(* IEC 61131-3 sources: Summary-ETFA22/ahorn/benchmark/Arcade, 15 files *)

(* ---- 4.4.SafeMotionIO.st ---- *)
PROGRAM SafeMotionIO
USING PLCopenX;

  VAR_INPUT
	S1_S_EStopIn : SAFEBOOL;
    S2_S_AutoMode : SAFEBOOL;
    S2_S_SetupMode : SAFEBOOL;
    S4_S_EnableSwitchCh1 : SAFEBOOL;
    S4_S_EnableSwitchCh2 : SAFEBOOL;
    S5_S_GuardSwitch : SAFEBOOL;
    S7_S_GuardLock : SAFEBOOL;
    S0_Reset : BOOL;
    S8_UnlockGuard : BOOL;
    M1_S_AcknowledgeSS1 : SAFEBOOL;
    M1_S_AcknowledgeSafeMotion : SAFEBOOL;
  END_VAR
  VAR_OUTPUT
    S_SafeStop_M1 : SAFEBOOL;
    S_SafeMotion_M1 : SAFEBOOL;
    S_Enable_M1 : SAFEBOOL;
    S_UnlockGuard_K1 : SAFEBOOL;
  END_VAR
  VAR
    S_SetupMode : SAFEBOOL;
    S_AutoMode : SAFEBOOL;
    S_SafeStandstill : SAFEBOOL;
    S_SafeMotionActive : SAFEBOOL;
    SF_EmergencyStop_1 : SF_EmergencyStopX;
  	SF_SafetyRequest_1 : SF_SafetyRequestX;
  	SF_SafetyRequest_2 : SafetyRequest_dummy;
  	SF_ModeSelector_1 : SF_ModeSelectorX;
  	SF_GuardLocking_1 : SF_GuardLockingX;
  	SF_EnableSwitch_1 : SF_EnableSwitchX;
  END_VAR

  SF_EmergencyStop_1(TRUE, S1_S_EStopIn, FALSE, FALSE, S0_Reset);
  SF_SafetyRequest_1(TRUE, SF_EmergencyStop_1.S_EstopOut, M1_S_AcknowledgeSS1, T#100ms, S0_Reset);
  SF_SafetyRequest_2(TRUE, S_AutoMode, M1_S_AcknowledgeSafeMotion, T#100ms, S0_Reset);
  SF_ModeSelector_1(TRUE, S2_S_AutoMode, S2_S_SetupMode, FALSE, FALSE, FALSE, FALSE, FALSE, FALSE, TRUE, FALSE, TRUE, T#50ms, S0_Reset);
  SF_GuardLocking_1(TRUE, S5_S_GuardSwitch, S_SafeStandstill OR S_SafeMotionActive, S7_S_GuardLock, S8_UnlockGuard, FALSE, FALSE, S0_Reset);
  SF_EnableSwitch_1(TRUE, S_SafeMotionActive AND S_SetupMode, S4_S_EnableSwitchCh1, S4_S_EnableSwitchCh2, FALSE, S0_Reset);

  S_SafeStandstill := SF_SafetyRequest_1.S_SafetyActive;
  S_SafeStop_M1 := SF_SafetyRequest_1.S_SafetyRequest;
  S_SafeMotionActive := SF_SafetyRequest_2.S_SafetyActive;
  S_SafeMotion_M1 := SF_SafetyRequest_2.S_SafetyRequest;
  S_SetupMode := SF_ModeSelector_1.S_Mode1Sel;
  S_AutoMode := SF_ModeSelector_1.S_Mode0Sel AND SF_GuardLocking_1.S_GuardLocked;
  S_UnlockGuard_K1 := SF_GuardLocking_1.S_UnlockGuard;
  S_Enable_M1 := SF_EnableSwitch_1.S_EnableSwitchOut;

END_PROGRAM

FUNCTION_BLOCK SafetyRequest_dummy
VAR_INPUT
        Activate        : BOOL;
        S_OpMode        : SAFEBOOL;
        S_Acknowledge   : SAFEBOOL;
        MonitoringTime  : TIME := T#0s;
        Reset           : BOOL ;
 END_VAR

 VAR_OUTPUT
        Ready : BOOL ;
        S_SafetyActive : SAFEBOOL ;
        S_SafetyRequest : SAFEBOOL ;
        Error : BOOL ;
        DiagCode : WORD:=16#0000 ;
 END_VAR

VAR
        R_TRIGatReset: R_TRIG;
        T1: TONX;
END_VAR

R_TRIGatReset(CLK:=Reset);

IF NOT Activate THEN
    DiagCode := 16#0000;
ELSE

CASE DiagCode OF
16#0000:
    IF Activate THEN
        DiagCode := 16#8001;
    END_IF;
16#8000:
    IF NOT S_Acknowledge THEN
        DiagCode := 16#C002;
    ELSIF S_OpMode THEN
        DiagCode := 16#8012;
    END_IF;
16#8001:
    IF R_TRIGatReset.Q AND NOT S_Acknowledge THEN
        DiagCode := 16#8002;
    ELSIF R_TRIGatReset.Q AND S_Acknowledge THEN
        DiagCode := 16#8012;
    END_IF;
16#8002:
    IF NOT S_OpMode THEN
        DiagCode := 16#8003;
    ELSIF S_Acknowledge THEN
        DiagCode := 16#8012;
    END_IF;
16#8003:
    IF T1.Q THEN
        DiagCode := 16#C003;
    ELSIF S_OpMode THEN
        DiagCode := 16#8012;
    ELSIF S_Acknowledge THEN
        DiagCode := 16#8000;
    END_IF;
16#8005:
    IF S_OpMode THEN
        DiagCode := 16#8012;
    END_IF;
16#8012:
    IF NOT S_Acknowledge THEN
        DiagCode := 16#8002;
    ELSIF NOT S_OpMode THEN
        DiagCode := 16#8003;
    END_IF;
16#C002:
    IF Reset AND NOT R_TRIGatReset.Q THEN
        DiagCode := 16#C004;
    ELSIF R_TRIGatReset.Q THEN
        DiagCode := 16#8005;
    END_IF;
16#C003:
    IF Reset AND NOT R_TRIGatReset.Q THEN
        DiagCode := 16#C005;
    ELSIF R_TRIGatReset.Q THEN
        DiagCode := 16#8005;
    END_IF;
16#C004:
    IF NOT Reset THEN
        DiagCode := 16#C002;
    END_IF;
16#C005:
    IF NOT Reset THEN
        DiagCode := 16#C003;
    END_IF;
END_CASE;
END_IF;

IF DiagCode <> 16#8003 THEN
    T1(IN:=false, PT:=MonitoringTime);
ELSE
	T1(IN:=true, PT:=MonitoringTime);
END_IF;

CASE DiagCode OF
16#0000:
    Ready := FALSE;
    S_SafetyActive := FALSE;
    S_SafetyRequest := FALSE;
    Error := FALSE;
16#8000:
    Ready := TRUE;
    S_SafetyActive := TRUE;
    S_SafetyRequest := FALSE;
    Error := FALSE;
16#8001:
    Ready := TRUE;
    S_SafetyActive := FALSE;
    S_SafetyRequest := FALSE;
    Error := FALSE;
16#8002:
    Ready := TRUE;
    S_SafetyActive := FALSE;
    S_SafetyRequest := TRUE;
    Error := FALSE;
16#8003:
    Ready := TRUE;
    S_SafetyActive := FALSE;
    S_SafetyRequest := FALSE;
    Error := FALSE;
16#8005:
    Ready := TRUE;
    S_SafetyActive := FALSE;
    S_SafetyRequest := FALSE;
    Error := FALSE;
16#8012:
    Ready := TRUE;
    S_SafetyActive := FALSE;
    S_SafetyRequest := TRUE;
    Error := FALSE;
16#C002:
    Ready := TRUE;
    S_SafetyActive := FALSE;
    S_SafetyRequest := FALSE;
    Error := TRUE;
16#C003:
    Ready := TRUE;
    S_SafetyActive := FALSE;
    S_SafetyRequest := FALSE;
    Error := TRUE;
16#C004:
    Ready := TRUE;
    S_SafetyActive := FALSE;
    S_SafetyRequest := FALSE;
    Error := TRUE;
16#C005:
    Ready := TRUE;
    S_SafetyActive := FALSE;
    S_SafetyRequest := FALSE;
    Error := TRUE;
END_CASE;

END_FUNCTION_BLOCK;

(* ---- antivalentX.st ---- *)
FUNCTION_BLOCK SF_Antivalent2
 VAR_INPUT
        Activate           : BOOL;
        S_ChannelNC        : SAFEBOOL;
        S_ChannelNO        : SAFEBOOL;
        DiscrepancyTime    : TIME;
 END_VAR
 VAR_OUTPUT
        Ready              : BOOL;
        S_AntivalentOut    : BOOL;
        Error              : BOOL;
        DiagCode           : WORD;
 END_VAR
 VAR
        T_1        : TONX;
 END_VAR

IF NOT Activate THEN
    DiagCode := 16#0000;
ELSE

CASE DiagCode OF
16#0000:
    IF Activate THEN
        DiagCode := 16#8001;
    END_IF;
16#8001:
    IF S_ChannelNC AND S_ChannelNO THEN
        DiagCode := 16#8004;
        T_1(IN:=1, PT:=DiscrepancyTime);
    ELSIF NOT S_ChannelNC AND NOT S_ChannelNO THEN
        DiagCode := 16#8014;
        T_1(IN:=1, PT:=DiscrepancyTime);
    ELSIF S_ChannelNC AND NOT S_ChannelNO THEN
        DiagCode := 16#8000;
    END_IF;
16#8004:
    IF T_1.Q THEN
        DiagCode := 16#C001;
    ELSIF NOT S_ChannelNC THEN
        DiagCode := 16#8001;
    ELSIF NOT S_ChannelNO THEN
        DiagCode := 16#8000;
    END_IF;
16#C001,
16#C002:
    IF NOT S_ChannelNC AND S_ChannelNO THEN
        DiagCode := 16#8001;
    END_IF;
16#8014:
    IF T_1.Q THEN
        DiagCode := 16#C002;
    ELSIF S_ChannelNO THEN
        DiagCode := 16#8001;
    ELSIF S_ChannelNC THEN
        DiagCode := 16#8000;
    END_IF;
16#C003:
    IF NOT S_ChannelNC AND S_ChannelNO THEN
        DiagCode := 16#8001;
    END_IF;
16#8005:
    IF T_1.Q THEN
        DiagCode := 16#C003;
    ELSIF NOT S_ChannelNC AND S_ChannelNO THEN
        DiagCode := 16#8001;
    END_IF;
16#8000:
    IF NOT S_ChannelNC OR S_ChannelNO THEN
        DiagCode := 16#8005;
        T_1(IN:=1, PT:=DiscrepancyTime);
    ELSIF NOT S_ChannelNC AND S_ChannelNO THEN
        DiagCode := 16#8001;
    END_IF;
END_CASE;
END_IF;

CASE DiagCode OF
16#0000:
    T_1(IN:=0, PT:=DiscrepancyTime);
    Ready := FALSE;
    Error := FALSE;
    S_AntivalentOut:= FALSE;
16#8000:
    T_1(IN:=0, PT:=DiscrepancyTime);
    Ready := TRUE;
    Error := FALSE;
    S_AntivalentOut := TRUE;
16#8001:
    T_1(IN:=0, PT:=DiscrepancyTime);
    Ready := TRUE;
    Error := FALSE;
    S_AntivalentOut:= FALSE;
16#8004,
16#8014,
16#8005:
	T_1(IN:=1, PT:=DiscrepancyTime);
    Ready := TRUE;
    Error := FALSE;
    S_AntivalentOut:= FALSE;
16#C001,
16#C002,
16#C003:
    T_1(IN:=0, PT:=DiscrepancyTime);
    Ready := TRUE;
    Error := TRUE;
    S_AntivalentOut:= FALSE;
END_CASE;

END_FUNCTION_BLOCK

(* ---- emergencyStopX.st ---- *)
FUNCTION_BLOCK SF_EmergencyStop2
VAR_INPUT
        Activate      : BOOL;
        S_EStopIn     : BOOL;
        S_StartReset  : BOOL;
        S_AutoReset   : BOOL;
        Reset         : BOOL;
 END_VAR

 VAR_OUTPUT
        Ready         : BOOL;
        S_EStopOut    : BOOL;
        Error         : BOOL;
        DiagCode      : WORD;
 END_VAR

 VAR
        R_TRIGatReset: R_TRIG;
 END_VAR

R_TRIGatReset(CLK:=Reset);

IF NOT Activate THEN
    DiagCode := 16#0000;
ELSE

CASE DiagCode OF
16#0000:
    IF Activate THEN
        DiagCode := 16#8001;
    END_IF;
16#8001:
    IF NOT S_StartReset THEN
        DiagCode := 16#8002;
    ELSIF S_StartReset AND NOT S_EStopIn THEN
        DiagCode := 16#8004;
    ELSIF S_EStopIn AND S_StartReset THEN
        DiagCode := 16#8000;
    END_IF;
16#8002:
    IF S_EStopIn THEN
        DiagCode := 16#8003;
    END_IF;
16#8003:
    IF Reset AND NOT R_TRIGatReset.Q THEN
        DiagCode := 16#C001;
    ELSIF NOT S_EStopIn THEN
        DiagCode := 16#8002;
    ELSIF R_TRIGatReset.Q THEN
        DiagCode := 16#8000;
    END_IF;
16#C001:
    IF NOT Reset THEN
        DiagCode := 16#8003;
    END_IF;
16#8004:
    IF S_EStopIn AND NOT S_AutoReset THEN
        DiagCode := 16#8005;
    ELSIF S_EStopIn AND S_AutoReset THEN
        DiagCode := 16#8000;
    END_IF;
16#8005:
    IF Reset AND NOT R_TRIGatReset.Q THEN
        DiagCode := 16#C002;
    ELSIF NOT S_EStopIn THEN
        DiagCode := 16#8004;
    ELSIF R_TRIGatReset.Q OR S_AutoReset THEN
        DiagCode := 16#8000;
    END_IF;
16#C002:
    IF NOT Reset THEN
        DiagCode := 16#8005;
    END_IF;
16#8000:
    IF NOT S_EStopIn THEN
        DiagCode := 16#8004;
    END_IF;
END_CASE;
END_IF;

CASE DiagCode OF
16#0000:
    Ready := FALSE;
    Error := FALSE;
    S_EStopOut := FALSE;
16#8001:
    Ready := TRUE;
    Error := FALSE;
    S_EStopOut := FALSE;
16#8002:
    Ready := TRUE;
    Error := FALSE;
    S_EStopOut := FALSE;
16#8003:
    Ready := TRUE;
    Error := FALSE;
    S_EStopOut := FALSE;
16#C001:
    Ready := TRUE;
    Error := TRUE;
    S_EStopOut := FALSE;
16#8004:
    Ready := TRUE;
    Error := FALSE;
    S_EStopOut := FALSE;
16#8005:
    Ready := TRUE;
    Error := FALSE;
    S_EStopOut := FALSE;
16#C002:
    Ready := TRUE;
    Error := TRUE;
    S_EStopOut := FALSE;
16#8000:
    Ready := TRUE;
    Error := FALSE;
    S_EStopOut := TRUE;
END_CASE;

END_FUNCTION_BLOCK

(* ---- enableSwitchX.st ---- *)
FUNCTION_BLOCK SF_EnableSwitch2
VAR_INPUT
	Activate          : BOOL := FALSE;
	S_SafetyActive    : SAFEBOOL := FALSE;
	S_EnableSwitchCh1 : SAFEBOOL := FALSE;
	S_EnableSwitchCh2 : SAFEBOOL := FALSE;
	S_AutoReset       : SAFEBOOL := FALSE;
	Reset             : BOOL := FALSE;
END_VAR

VAR_OUTPUT
	Ready: BOOL := FALSE;
	S_EnableSwitchOut: SAFEBOOL := FALSE;
	Error: BOOL := FALSE;
	DiagCode: WORD := 16#0000;
END_VAR

VAR
	R_TRIGatReset: R_TRIG;
END_VAR

R_TRIGatReset(CLK:=Reset);

IF NOT Activate THEN
    DiagCode := 16#0000;
ELSIF NOT S_SafetyActive THEN
    DiagCode := 16#8004;
ELSE

CASE DiagCode OF
16#0000:
    IF Activate THEN
	DiagCode := 16#8004;
    END_IF;

16#8000:
	IF (NOT (S_EnableSwitchCh1 OR S_EnableSwitchCh2)) OR (S_EnableSwitchCh1 AND NOT S_EnableSwitchCh2) THEN
		DiagCode := 16#8007;
	ELSIF NOT S_EnableSwitchCh1 AND S_EnableSwitchCh2 THEN
		DiagCode := 16#8006;
	END_IF;

16#8004:
    IF S_SafetyActive THEN
		DiagCode := 16#8005;
	END_IF;

16#8005:
	IF NOT (NOT S_EnableSwitchCh1 AND S_EnableSwitchCh2) THEN
		DiagCode := 16#C010;
	ELSIF NOT S_EnableSwitchCh1 AND S_EnableSwitchCh2 THEN
		DiagCode := 16#8006;
	END_IF;

16#8006:
	IF S_EnableSwitchCh1 AND S_EnableSwitchCh2 THEN
		DiagCode := 16#8000;
	ELSIF (NOT (S_EnableSwitchCh1 OR S_EnableSwitchCh2)) OR (S_EnableSwitchCh1 AND NOT S_EnableSwitchCh2) THEN
		DiagCode := 16#8007;
	END_IF;

16#8007:
	IF S_EnableSwitchCh1 AND S_EnableSwitchCh2 THEN
		DiagCode := 16#C030;
	ELSIF NOT S_EnableSwitchCh1 AND S_EnableSwitchCh2 THEN
		DiagCode := 16#8006;
	END_IF;
16#C001:
	IF NOT Reset THEN
		DiagCode := 16#C020;
	END_IF;
16#C002:
	IF NOT Reset THEN
		DiagCode := 16#C040;
	END_IF;
16#C010:
	IF NOT S_EnableSwitchCh1 AND S_EnableSwitchCh2 THEN
		DiagCode := 16#C020;
	END_IF;

16#C020:
	IF NOT (NOT S_EnableSwitchCh1 AND S_EnableSwitchCh2) THEN
		DiagCode := 16#C010;
	ELSIF Reset AND NOT R_TRIGatReset.Q AND NOT S_AutoReset THEN
		DiagCode := 16#C001;
	ELSIF R_TRIGatReset.Q OR S_AutoReset THEN
		DiagCode := 16#8006;
	END_IF;

16#C030:
	IF NOT (S_EnableSwitchCh1 AND S_EnableSwitchCh2) THEN
		DiagCode := 16#C040;
	END_IF;

16#C040:
	IF S_EnableSwitchCh1 AND S_EnableSwitchCh2 THEN
		DiagCode := 16#C030;
	ELSIF Reset AND R_TRIGatReset.Q AND NOT S_AutoReset THEN
		DiagCode := 16#C002;
	ELSIF R_TRIGatReset.Q OR S_AutoReset THEN
		DiagCode := 16#8007;
	END_IF;
END_CASE;

END_IF;

CASE DiagCode OF
16#C001,
16#C002,
16#C010,
16#C020,
16#C030,
16#C040:
	Ready := TRUE;
	S_EnableSwitchOut := FALSE;
	Error := TRUE;
16#0000:
	Ready := FALSE;
	S_EnableSwitchOut := FALSE;
	Error := FALSE;
16#8000:
	Ready := TRUE;
	S_EnableSwitchOut := TRUE;
	Error := FALSE;

16#8004,
16#8005,
16#8006,
16#8007:
	Ready := TRUE;
	S_EnableSwitchOut := FALSE;
	Error := FALSE;

END_CASE;

END_FUNCTION_BLOCK

(* ---- equivalentX.st ---- *)
FUNCTION_BLOCK equivalentX
VAR_INPUT
	Activate		: BOOL;
	S_ChannelA		: BOOL;
	S_ChannelB		: BOOL;
	DiscrepancyTime 	: TIME;
END_VAR
VAR_OUTPUT
	Ready		: BOOL;
	S_EquivalentOut	: BOOL;
	Error		: BOOL;
	DiagCode	: WORD;
END_VAR
VAR
 DiscrepancyTimer	: TONX;
END_VAR

IF NOT Activate THEN
    DiagCode := 16#0000;
ELSE

CASE DiagCode OF
16#0000:
    IF Activate THEN
	DiagCode := 16#8001;
    END_IF;
16#8001:
    IF S_ChannelA AND NOT S_ChannelB THEN
	DiagCode := 16#8004;
    ELSIF S_ChannelB AND NOT S_ChannelA THEN
	DiagCode := 16#8014;
    ELSIF S_ChannelA AND S_ChannelB THEN
	DiagCode := 16#8000;
    END_IF;
16#8004:
    IF DiscrepancyTimer.Q THEN
	DiagCode := 16#C001;
    ELSIF NOT S_ChannelA THEN
	DiagCode := 16#8001;
    ELSIF S_ChannelB THEN
	DiagCode := 16#8000;
    END_IF;
16#C001,
16#C002:
    IF NOT S_ChannelA AND NOT S_ChannelB THEN
	DiagCode := 16#8001;
    END_IF;
16#8014:
    IF DiscrepancyTimer.Q THEN
	DiagCode := 16#C002;
    ELSIF NOT S_ChannelB THEN
	DiagCode := 16#8001;
    ELSIF S_ChannelA THEN
	DiagCode := 16#8000;
    END_IF;
16#C003:
    IF NOT S_ChannelA AND NOT S_ChannelB THEN
	DiagCode := 16#8001;
    END_IF;
16#8005:
    IF DiscrepancyTimer.Q THEN
	DiagCode := 16#C003;
    ELSIF NOT S_ChannelA AND NOT S_ChannelB THEN
	DiagCode := 16#8001;
    END_IF;
16#8000:
    IF S_ChannelA XOR S_ChannelB THEN
	DiagCode := 16#8005;
    ELSIF NOT S_ChannelA AND NOT S_ChannelB THEN
	DiagCode := 16#8001;
    END_IF;
END_CASE;

END_IF;

CASE DiagCode OF
16#0000:
    DiscrepancyTimer(IN:=0, PT:=DiscrepancyTime);
    Ready := FALSE;
    Error := FALSE;
    S_EquivalentOut:= FALSE;
16#8000:
    DiscrepancyTimer(IN:=0, PT:=DiscrepancyTime);
    Ready := TRUE;
    Error := FALSE;
    S_EquivalentOut := TRUE;
16#8001:
    DiscrepancyTimer(IN:=0, PT:=DiscrepancyTime);
    Ready := TRUE;
    Error := FALSE;
    S_EquivalentOut:= FALSE;
16#8004,
16#8014,
16#8005:
	DiscrepancyTimer(IN:=1, PT:=DiscrepancyTime);
    Ready := TRUE;
    Error := FALSE;
    S_EquivalentOut:= FALSE;
16#C001,
16#C002,
16#C003:
    DiscrepancyTimer(IN:=0, PT:=DiscrepancyTime);
    Ready := TRUE;
    Error := TRUE;
    S_EquivalentOut:= FALSE;
END_CASE;

END_FUNCTION_BLOCK

(* ---- guardLockingX.st ---- *)
FUNCTION_BLOCK SF_GuardLocking2
VAR_INPUT
        Activate          : BOOL;
        S_GuardMonitoring : SAFEBOOL;
        S_SafetyActive    : SAFEBOOL;
        S_GuardLock       : SAFEBOOL;
        UnlockRequest     : BOOL;
        S_StartReset      : SAFEBOOL;
        S_AutoReset       : SAFEBOOL;
        Reset             : BOOL;
 END_VAR

 VAR_OUTPUT
    Ready             : BOOL;
    S_GuardLocked     : SAFEBOOL;
    S_UnlockGuard     : SAFEBOOL;
    Error             : BOOL;
         DiagCode                  : WORD:=16#0000;
 END_VAR

VAR
        R_TRIGatReset: R_TRIG;
        R_TRIGatUnlockRequest: R_TRIG;
END_VAR

R_TRIGatReset(CLK:=Reset);
R_TRIGatUnlockRequest(CLK:=UnlockRequest);

IF NOT Activate THEN
    DiagCode := 16#0000;
END_IF;

CASE DiagCode OF
16#0000:
    IF Activate THEN
        DiagCode := 16#8001;
    END_IF;
16#8000:
    IF NOT S_GuardLock OR NOT S_GuardMonitoring THEN
        DiagCode := 16#C004;
    ELSIF R_TRIGatUnlockRequest.Q AND S_SafetyActive THEN
        DiagCode := 16#8013;
    END_IF;
16#8001:
    IF Reset AND NOT R_TRIGatReset.Q AND NOT S_StartReset THEN
        DiagCode := 16#C001;
    ELSIF NOT S_GuardLock OR NOT S_GuardMonitoring THEN
        DiagCode := 16#8011;
    ELSIF (R_TRIGatReset.Q OR S_StartReset) AND S_GuardMonitoring AND S_GuardLock THEN
        DiagCode := 16#8000;
    END_IF;
16#8003:
    IF Reset AND NOT R_TRIGatReset.Q AND NOT S_AutoReset THEN
        DiagCode := 16#C003;
    ELSIF NOT S_GuardMonitoring OR NOT S_GuardLock THEN
        DiagCode := 16#8011;
    ELSIF R_TRIGatReset.Q OR S_AutoReset THEN
        DiagCode := 16#8000;
    END_IF;
16#8011:
    IF NOT S_SafetyActive AND (NOT S_GuardMonitoring OR NOT S_GuardLock) THEN
        DiagCode := 16#C004;
    ELSIF (S_SafetyActive AND UnlockRequest) OR NOT S_GuardMonitoring THEN
        DiagCode := 16#8012;
    ELSIF S_GuardMonitoring AND S_GuardLock THEN
        DiagCode := 16#8003;
    END_IF;
16#8012:
    IF S_GuardMonitoring THEN
        DiagCode := 16#8013;
    ELSIF NOT S_SafetyActive AND NOT S_GuardMonitoring THEN
        DiagCode := 16#C004;
    END_IF;
16#8013:
    IF NOT S_GuardMonitoring THEN
        DiagCode := 16#8012;
    ELSIF NOT UnlockRequest THEN
        DiagCode := 16#8011;
    END_IF;
16#8014:
    IF Reset AND NOT R_TRIGatReset.Q THEN
        DiagCode := 16#C002;
    ELSIF NOT S_SafetyActive THEN
        DiagCode := 16#C004;
    ELSIF R_TRIGatReset.Q THEN
        DiagCode := 16#8011;
    END_IF;
16#C001:
    IF NOT Reset THEN
        DiagCode := 16#8001;
    END_IF;
16#C002:
    IF NOT Reset THEN
        DiagCode := 16#8014;
    END_IF;
16#C003:
    IF NOT Reset THEN
        DiagCode := 16#8003;
    END_IF;
16#C004:
    IF S_SafetyActive THEN
        DiagCode := 16#8014;
    END_IF;
END_CASE;

CASE DiagCode OF
16#0000:
    Ready := FALSE;
    S_GuardLocked := FALSE;
    S_UnlockGuard := FALSE;
    Error := FALSE;
16#8000:
    Ready := TRUE;
    S_GuardLocked := TRUE;
    S_UnlockGuard := FALSE;
    Error := FALSE;
16#8001,
16#8003,
16#8011,
16#8014:
    Ready := TRUE;
    S_GuardLocked := FALSE;
    S_UnlockGuard := FALSE;
    Error := FALSE;
16#8012,
16#8013:
    Ready := TRUE;
    S_GuardLocked := FALSE;
    S_UnlockGuard := TRUE;
    Error := FALSE;
16#C001,
16#C002,
16#C003,
16#C004:
    Ready := TRUE;
    S_GuardLocked := FALSE;
    S_UnlockGuard := FALSE;
    Error := TRUE;
END_CASE;

END_FUNCTION_BLOCK

(* ---- guardMonitoringX.st ---- *)
FUNCTION_BLOCK SF_GuardMonitoring2
VAR_INPUT
        Activate        : BOOL := FALSE;
        S_GuardSwitch1  : SAFEBOOL := FALSE;
        S_GuardSwitch2  : SAFEBOOL := FALSE;
        DiscrepancyTime : TIME := T#0s;
        S_StartReset    : SAFEBOOL := FALSE;
        S_AutoReset     : SAFEBOOL := FALSE;
        Reset           : BOOL := FALSE;
END_VAR
VAR_OUTPUT
        Ready             : BOOL := FALSE;
        S_GuardMonitoring : BOOL := FALSE;
        Error             : BOOL := FALSE;
        DiagCode          : WORD := 16#0000;
END_VAR
VAR
    R_TRIGatReset : R_TRIG;
    DiscrepancyTimer : TONX;
END_VAR

R_TRIGatReset(CLK:=Reset);

IF NOT Activate THEN
    DiagCode := 16#0000;
ELSE

CASE DiagCode OF
16#0000:
    IF Activate THEN
        DiagCode := 16#8001;
    END_IF;
16#8001:
    IF NOT S_GuardSwitch1 OR NOT S_GuardSwitch2 THEN
        DiagCode := 16#8002;
    ELSIF S_GuardSwitch1 AND S_GuardSwitch2 AND NOT S_StartReset THEN
        DiagCode := 16#8003;
    ELSIF S_GuardSwitch1 AND S_GuardSwitch2 AND S_StartReset THEN
        DiagCode := 16#8000;
    END_IF;
16#8002:
    IF NOT S_GuardSwitch1 AND NOT S_GuardSwitch2 THEN
        DiagCode := 16#8012;
    END_IF;
16#8003:
    IF Reset AND NOT R_TRIGatReset.Q THEN
        DiagCode := 16#C001;
    ELSIF NOT S_GuardSwitch1 OR NOT S_GuardSwitch2 THEN
        DiagCode := 16#8002;
    ELSIF R_TRIGatReset.Q THEN
        DiagCode := 16#8000;
    END_IF;
16#8012:
    IF S_GuardSwitch1 THEN
        DiagCode := 16#8004;
    ELSIF S_GuardSwitch2 THEN
        DiagCode := 16#8014;
    END_IF;
16#8004:
    IF DiscrepancyTimer.Q THEN
        DiagCode := 16#C011;
    ELSIF NOT S_GuardSwitch1 THEN
        DiagCode := 16#8002;
    ELSIF S_GuardSwitch2 THEN
        DiagCode := 16#8005;
    END_IF;
16#8014:
    IF DiscrepancyTimer.Q THEN
        DiagCode := 16#C012;
    ELSIF NOT S_GuardSwitch2 THEN
        DiagCode := 16#8002;
    ELSIF S_GuardSwitch1 THEN
        DiagCode := 16#8005;
    END_IF;
16#8005:
    IF NOT S_GuardSwitch1 OR NOT S_GuardSwitch2 THEN
        DiagCode := 16#8002;
    ELSIF NOT S_AutoReset THEN
        DiagCode := 16#8003;
    ELSIF S_AutoReset THEN
        DiagCode := 16#8000;
    END_IF;
16#8000:
    IF NOT S_GuardSwitch1 OR NOT S_GuardSwitch2 THEN
        DiagCode := 16#8002;
    END_IF;
16#C001:
    IF NOT Reset THEN
        DiagCode := 16#8003;
    END_IF;
16#C011:
    IF NOT S_GuardSwitch1 AND NOT S_GuardSwitch2 THEN
        DiagCode := 16#8012;
    END_IF;
16#C012:
    IF NOT S_GuardSwitch1 AND NOT S_GuardSwitch2 THEN
        DiagCode := 16#8012;
    END_IF;
END_CASE;
END_IF;

CASE DiagCode OF
16#0000:
    DiscrepancyTimer(IN:=FALSE, PT:=DiscrepancyTime);
    Ready := FALSE;
    Error := FALSE;
    S_GuardMonitoring := FALSE;
16#8000:
    DiscrepancyTimer(IN:=FALSE, PT:=DiscrepancyTime);
    Ready := TRUE;
    Error := FALSE;
    S_GuardMonitoring  := TRUE;
16#8001,
16#8002,
16#8003,
16#8012,
16#8005:
    DiscrepancyTimer(IN:=FALSE, PT:=DiscrepancyTime);
    Ready := TRUE;
    Error := FALSE;
    S_GuardMonitoring := FALSE;
16#8004,
16#8014:
	DiscrepancyTimer(IN:=TRUE, PT:=DiscrepancyTime);
    Ready := TRUE;
    Error := FALSE;
    S_GuardMonitoring := FALSE;
16#C001,
16#C011,
16#C012:
    DiscrepancyTimer(IN:=FALSE, PT:=DiscrepancyTime);
    Ready := TRUE;
    Error := TRUE;
    S_GuardMonitoring := FALSE;
END_CASE;

END_FUNCTION_BLOCK

(* ---- ModeSelectorX.st ---- *)
FUNCTION_BLOCK ModeSelectorX
VAR_INPUT
        Activate        : BOOL;
        S_Mode0         : BOOL;
        S_Mode1         : BOOL;
        S_Mode2         : BOOL;
        S_Mode3         : BOOL;
        S_Mode4         : BOOL;
        S_Mode5         : BOOL;
        S_Mode6         : BOOL;
        S_Mode7         : BOOL;
        S_Unlock        : BOOL;
        S_SetMode       : BOOL;
        AutoSetMode     : BOOL;
        ModeMonitorTime : TIME;
        Reset           : BOOL;
 END_VAR
 VAR_OUTPUT
        Ready           : BOOL;
        S_Mode0Sel      : BOOL;
        S_Mode1Sel      : BOOL;
        S_Mode2Sel      : BOOL;
        S_Mode3Sel      : BOOL;
        S_Mode4Sel      : BOOL;
        S_Mode5Sel      : BOOL;
        S_Mode6Sel      : BOOL;
        S_Mode7Sel      : BOOL;
        S_AnyModeSel    : BOOL;
        Error           : BOOL;
        DiagCode        : WORD;
 END_VAR
 VAR
        T_1        : TONX;                 (* Timer for S2, transition T27 *)
 END_VAR

 VAR
        R_TRIGatReset: R_TRIG;
        R_TRIGatSetMode: R_TRIG;
        F_TRIGatModeSel0: F_TRIG;
        R_TRIGatModeSel0: R_TRIG;
        fallingEdgeDetected : BOOL;
 END_VAR

 VAR_TEMP
    Error1 : BOOL;
    Error2 : BOOL;
 END_VAR

R_TRIGatReset(CLK:=Reset);
R_TRIGatSetMode(CLK:=S_SetMode);

IF NOT Activate THEN
    DiagCode := 16#0000;
ELSE

IF (S_Mode0 + S_Mode1 + S_Mode2 + S_Mode3 + S_Mode4 + S_Mode5 + S_Mode6 + S_Mode7 > 1) THEN
    Error1 := true;
ELSE
    Error1 := false;
END_IF;

CASE DiagCode OF
16#0000:
    IF Activate THEN
        DiagCode := 16#8005;
    END_IF;
16#8005:
    IF (NOT S_Mode0 AND NOT S_Mode1 AND NOT S_Mode2 AND NOT S_Mode3 AND NOT S_Mode4 AND NOT S_Mode5 AND NOT S_Mode6 AND NOT S_Mode7) THEN
        F_TRIGatModeSel0(CLK:=false);
        R_TRIGatModeSel0(CLK:=false);
    ELSE
        F_TRIGatModeSel0(CLK:=true);
        R_TRIGatModeSel0(CLK:=true);
    END_IF;

    IF F_TRIGatModeSel0.Q THEN
        fallingEdgeDetected := TRUE;
    END_IF;

    IF fallingEdgeDetected THEN
        T_1(IN:=true, PT:=ModeMonitorTime);
    ELSIF R_TRIGatModeSel0.Q THEN
        T_1(IN:=false, PT:=ModeMonitorTime);
        fallingEdgeDetected := FALSE;
    END_IF;

    Error2 := T_1.Q;

    IF Error1 THEN
        DiagCode := 16#C001;
    ELSIF Error2 THEN
        DiagCode := 16#C002;
    ELSIF ((AutoSetMode OR R_TRIGatSetMode.Q) AND S_Unlock AND (S_Mode0 + S_Mode1 + S_Mode2 + S_Mode3 + S_Mode4 + S_Mode5 + S_Mode6 + S_Mode7 = 1)) THEN
        DiagCode := 16#8000;
    END_IF;
16#8000:
    IF Error1 THEN
        DiagCode := 16#C001;
    ELSIF (S_Mode0 <> S_Mode0Sel OR S_Mode1 <> S_Mode1Sel OR S_Mode2 <> S_Mode2Sel OR S_Mode3 <> S_Mode3Sel
          OR S_Mode4 <> S_Mode4Sel OR S_Mode5 <> S_Mode5Sel OR S_Mode6 <> S_Mode6Sel OR S_Mode7 <> S_Mode7Sel) THEN
        DiagCode := 16#8005;
        fallingEdgeDetected := FALSE;
    ELSIF (NOT S_Unlock) THEN
        DiagCode := 16#8004;
    END_IF;
16#8004:
    IF S_Unlock THEN
        DiagCode := 16#8000;
    END_IF;
16#C001:
    IF Reset AND NOT R_TRIGatReset.Q THEN
        DiagCode := 16#C003;
    ELSIF R_TRIGatReset.Q THEN
        DiagCode := 16#8005;
        fallingEdgeDetected := FALSE;
    END_IF;
16#C002:
    IF Reset AND NOT R_TRIGatReset.Q THEN
        DiagCode := 16#C004;
    ELSIF R_TRIGatReset.Q THEN
        DiagCode := 16#8005;
        fallingEdgeDetected := FALSE;
    END_IF;
16#C003:
    IF (NOT Reset) THEN
                DiagCode := 16#C001;
    END_IF;
16#C004:
    IF (NOT Reset) THEN
                DiagCode := 16#C002;
    END_IF;
END_CASE;
END_IF;

CASE DiagCode OF
16#0000:
    Ready := false;
    S_Mode0Sel := false;
    S_Mode1Sel := false;
    S_Mode2Sel := false;
    S_Mode3Sel := false;
    S_Mode4Sel := false;
    S_Mode5Sel := false;
    S_Mode6Sel := false;
    S_Mode7Sel := false;
    S_AnyModeSel := false;
    Error := false;
16#8005:
    Ready := true;
    S_Mode0Sel := false;
    S_Mode1Sel := false;
    S_Mode2Sel := false;
    S_Mode3Sel := false;
    S_Mode4Sel := false;
    S_Mode5Sel := false;
    S_Mode6Sel := false;
    S_Mode7Sel := false;
    S_AnyModeSel := false;
    Error := false;
16#8000:
    Ready := true;
    S_Mode0Sel := S_Mode0;
    S_Mode1Sel := S_Mode1;
    S_Mode2Sel := S_Mode2;
    S_Mode3Sel := S_Mode3;
    S_Mode4Sel := S_Mode4;
    S_Mode5Sel := S_Mode5;
    S_Mode6Sel := S_Mode6;
    S_Mode7Sel := S_Mode7;
    S_AnyModeSel := true;
    Error := false;
16#8004:
    Ready := true;
    S_AnyModeSel := true;
    Error := false;
16#C001,
16#C002,
16#C003,
16#C004:
    Ready := true;
    S_Mode0Sel := false;
    S_Mode1Sel := false;
    S_Mode2Sel := false;
    S_Mode3Sel := false;
    S_Mode4Sel := false;
    S_Mode5Sel := false;
    S_Mode6Sel := false;
    S_Mode7Sel := false;
    S_AnyModeSel := false;
    Error := true;
END_CASE;

IF (DiagCode <> 16#8005) THEN
    T_1(IN:=false, PT:=ModeMonitorTime);
END_IF;
END_FUNCTION_BLOCK

(* ---- safelyLimitSpeedX.st ---- *)
FUNCTION_BLOCK SF_SafelyLimitSpeed2
 VAR_INPUT
    Activate          : BOOL;
    S_OpMode          : SAFEBOOL;
    S_Enabled         : SAFEBOOL;
    AxisID            : INT;
    MonitoringTime    : TIME;
    Reset             : BOOL;
    Acknowledge       : BOOL;      (* This is an internal input *)
 END_VAR

 VAR_OUTPUT
    Ready             : BOOL;
    S_SafetyActive    : SAFEBOOL;
    Error             : BOOL;
    DiagCode          : WORD:=16#0000;
 END_VAR

 VAR
    R_TRIGatReset: R_TRIG;
    T_1: TONX;
 END_VAR

R_TRIGatReset(CLK:=Reset);

IF NOT Activate THEN
    DiagCode := 16#0000;
END_IF;

T_1(IN:=Activate AND NOT S_OpMode, PT:=MonitoringTime);

CASE DiagCode OF
16#0000:
    IF Activate THEN
        DiagCode := 16#8001;
    END_IF;
16#8000:
    IF NOT Acknowledge THEN
        DiagCode := 16#C002;
    ELSIF S_OpMode THEN
        DiagCode := 16#8012;
    ELSIF S_Enabled THEN
        DiagCode := 16#8004;
    END_IF;
16#8001:
    IF Reset AND NOT R_TRIGatReset.Q THEN
        DiagCode := 16#C001;
    ELSIF R_TRIGatReset.Q AND NOT Acknowledge THEN
        DiagCode := 16#8002;
    ELSIF R_TRIGatReset.Q AND Acknowledge THEN
        DiagCode := 16#8012;
    END_IF;
16#8002:
    IF NOT S_OpMode THEN
        DiagCode := 16#8003;
    ELSIF Acknowledge THEN
        DiagCode := 16#8012;
    END_IF;
16#8003:
    IF T_1.Q THEN
        DiagCode := 16#C003;
    ELSIF S_OpMode THEN
        DiagCode := 16#8012;
    ELSIF Acknowledge AND NOT S_Enabled THEN
        DiagCode := 16#8000;
    ELSIF Acknowledge AND S_Enabled THEN
        DiagCode := 16#8004;
    END_IF;
16#8004:
    IF NOT Acknowledge THEN
        DiagCode := 16#C002;
    ELSIF S_OpMode THEN
        DiagCode := 16#8012;
    ELSIF NOT S_Enabled THEN
        DiagCode := 16#8000;
    END_IF;
16#8005:
    IF S_OpMode THEN
        DiagCode := 16#8012;
    END_IF;
16#8012:
    IF NOT Acknowledge THEN
        DiagCode := 16#8002;
    ELSIF NOT S_OpMode THEN
        DiagCode := 16#8003;
    END_IF;
16#C001:
    IF NOT Reset THEN
        DiagCode := 16#8001;
    END_IF;
16#C002:
    IF Reset AND NOT R_TRIGatReset.Q THEN
        DiagCode := 16#C004;
    ELSIF R_TRIGatReset.Q THEN
        DiagCode := 16#8005;
    END_IF;
16#C003:
    IF Reset AND NOT R_TRIGatReset.Q THEN
        DiagCode := 16#C005;
    ELSIF R_TRIGatReset.Q THEN
        DiagCode := 16#8005;
    END_IF;
16#C004:
    IF NOT Reset THEN
        DiagCode := 16#C002;
    END_IF;
16#C005:
    IF NOT Reset THEN
        DiagCode := 16#C003;
    END_IF;
END_CASE;

CASE DiagCode OF
16#0000:
    Ready := FALSE;
    S_SafetyActive := FALSE;
    Error := FALSE;
16#8000,
16#8004:
    Ready := TRUE;
    S_SafetyActive := TRUE;
    Error := FALSE;
16#8001,
16#8002,
16#8003,
16#8005,
16#8012:
    Ready := TRUE;
    S_SafetyActive := FALSE;
    Error := FALSE;
16#C001,
16#C002,
16#C003,
16#C004,
16#C005:
    Ready := TRUE;
    S_SafetyActive := FALSE;
    Error := TRUE;
END_CASE;

END_FUNCTION_BLOCK

(* ---- safestopX.st ---- *)
FUNCTION_BLOCK safestopX
 VAR_INPUT
    Activate          : BOOL;
    S_StopIn          : SAFEBOOL;
    AxisID            : INT;
    MonitoringTime    : TIME;
    Reset             : BOOL;
    Acknowledge       : BOOL;      (* This is an internal input *)
 END_VAR

 VAR_OUTPUT
    Ready             : BOOL;
    S_Stopped         : SAFEBOOL;
    Error             : BOOL;
    DiagCode          : WORD:=16#0000;
 END_VAR

 VAR
    R_TRIGatReset: R_TRIG;
    T_1: DCTimer;
 END_VAR

R_TRIGatReset(CLK:=Reset);

IF NOT Activate THEN
    DiagCode := 16#0000;
ELSE

T_1(IN:=Activate AND NOT S_StopIn, PT:=MonitoringTime);

CASE DiagCode OF
16#0000:
    IF Activate THEN
        DiagCode := 16#8001;
    END_IF;
16#8000:
    IF NOT Acknowledge THEN
        DiagCode := 16#C002;
    ELSIF S_StopIn THEN
        DiagCode := 16#8012;
    END_IF;
16#8001:
    IF R_TRIGatReset.Q AND NOT Acknowledge THEN
        DiagCode := 16#8002;
    ELSIF R_TRIGatReset.Q AND Acknowledge THEN
        DiagCode := 16#8012;
    END_IF;
16#8002:
    IF NOT S_StopIn THEN
        DiagCode := 16#8003;
    ELSIF Acknowledge THEN
        DiagCode := 16#8012;
    END_IF;
16#8003:
    IF T_1.DiagCode = 1 THEN
        DiagCode := 16#C003;
    ELSIF S_StopIn THEN
        DiagCode := 16#8012;
    ELSIF Acknowledge THEN
        DiagCode := 16#8000;
    END_IF;
16#8005:
    IF S_StopIn THEN
        DiagCode := 16#8012;
    END_IF;
16#8012:
    IF NOT Acknowledge THEN
        DiagCode := 16#8002;
    ELSIF NOT S_StopIn THEN
        DiagCode := 16#8003;
    ELSIF Acknowledge THEN
        DiagCode := 16#8000;
    END_IF;
16#C002:
    IF Reset AND NOT R_TRIGatReset.Q THEN
        DiagCode := 16#C004;
    ELSIF R_TRIGatReset.Q THEN
        DiagCode := 16#8005;
    END_IF;
16#C003:
    IF Reset AND NOT R_TRIGatReset.Q THEN
        DiagCode := 16#C005;
    ELSIF R_TRIGatReset.Q THEN
        DiagCode := 16#8005;
    END_IF;
16#C004:
    IF NOT Reset THEN
        DiagCode := 16#C002;
    END_IF;
16#C005:
    IF NOT Reset THEN
        DiagCode := 16#C003;
    END_IF;
END_CASE;

END_IF;

CASE DiagCode OF
16#0000:
    Ready := FALSE;
    S_Stopped := FALSE;
    Error := FALSE;
16#8000:
    Ready := TRUE;
    S_Stopped := TRUE;
    Error := FALSE;
16#8001,
16#8002,
16#8003,
16#8005,
16#8012:
    Ready := TRUE;
    S_Stopped := FALSE;
    Error := FALSE;
16#C002,
16#C003,
16#C004,
16#C005:
    Ready := TRUE;
    S_Stopped := FALSE;
    Error := TRUE;
END_CASE;

END_FUNCTION_BLOCK

FUNCTION_BLOCK DCTimer
VAR_INPUT
  IN : BOOL;
  PT : TIME;
END_VAR
VAR
    running : BOOL;
END_VAR
VAR_TEMP
    timeout : BOOL;
END_VAR
VAR_OUTPUT
  DiagCode : WORD;
  ET : TIME;
END_VAR

  timeout := UNKNOWN_BOOL();

  IF NOT IN THEN
    DiagCode := 0;
    running := FALSE;
  ELSIF NOT running AND (DiagCode = 0) THEN
    running := TRUE;
  ELSIF running AND (DiagCode = 0) THEN
    IF timeout THEN
    	DiagCode := 1;
    	running := FALSE;
	ELSE
		DiagCode := 0;
		running := TRUE;
    END_IF;

  END_IF

  ET := UNKNOWN_TIME();
END_FUNCTION_BLOCK

(* ---- safetyRequestX.st ---- *)
FUNCTION_BLOCK SF_SafetyRequest2
VAR_INPUT
        Activate        : BOOL;
        S_OpMode        : SAFEBOOL;
        S_Acknowledge   : SAFEBOOL;
        MonitoringTime  : TIME := T#0s;
        Reset           : BOOL ;
 END_VAR

 VAR_OUTPUT
        Ready : BOOL ;
        S_SafetyActive : SAFEBOOL ;
        S_SafetyRequest : SAFEBOOL ;
        Error : BOOL ;
        DiagCode : WORD:=16#0000 ;
 END_VAR

VAR
        R_TRIGatReset: R_TRIG;
        T1: TONX;
END_VAR

R_TRIGatReset(CLK:=Reset);

IF NOT Activate THEN
    DiagCode := 16#0000;
ELSE

CASE DiagCode OF
16#0000:
    IF Activate THEN
        DiagCode := 16#8001;
    END_IF;
16#8000:
    IF NOT S_Acknowledge THEN
        DiagCode := 16#C002;
    ELSIF S_OpMode THEN
        DiagCode := 16#8012;
    END_IF;
16#8001:
    IF R_TRIGatReset.Q AND NOT S_Acknowledge THEN
        DiagCode := 16#8002;
    ELSIF R_TRIGatReset.Q AND S_Acknowledge THEN
        DiagCode := 16#8012;
    END_IF;
16#8002:
    IF NOT S_OpMode THEN
        DiagCode := 16#8003;
    ELSIF S_Acknowledge THEN
        DiagCode := 16#8012;
    END_IF;
16#8003:
    IF T1.Q THEN
        DiagCode := 16#C003;
    ELSIF S_OpMode THEN
        DiagCode := 16#8012;
    ELSIF S_Acknowledge THEN
        DiagCode := 16#8000;
    END_IF;
16#8005:
    IF S_OpMode THEN
        DiagCode := 16#8012;
    END_IF;
16#8012:
    IF NOT S_Acknowledge THEN
        DiagCode := 16#8002;
    ELSIF NOT S_OpMode THEN
        DiagCode := 16#8003;
    END_IF;
16#C002:
    IF Reset AND NOT R_TRIGatReset.Q THEN
        DiagCode := 16#C004;
    ELSIF R_TRIGatReset.Q THEN
        DiagCode := 16#8005;
    END_IF;
16#C003:
    IF Reset AND NOT R_TRIGatReset.Q THEN
        DiagCode := 16#C005;
    ELSIF R_TRIGatReset.Q THEN
        DiagCode := 16#8005;
    END_IF;
16#C004:
    IF NOT Reset THEN
        DiagCode := 16#C002;
    END_IF;
16#C005:
    IF NOT Reset THEN
        DiagCode := 16#C003;
    END_IF;
END_CASE;
END_IF;

IF DiagCode <> 16#8003 THEN
    T1(IN:=false, PT:=MonitoringTime);
ELSE
	T1(IN:=true, PT:=MonitoringTime);
END_IF;

CASE DiagCode OF
16#0000:
    Ready := FALSE;
    S_SafetyActive := FALSE;
    S_SafetyRequest := FALSE;
    Error := FALSE;
16#8000:
    Ready := TRUE;
    S_SafetyActive := TRUE;
    S_SafetyRequest := FALSE;
    Error := FALSE;
16#8001:
    Ready := TRUE;
    S_SafetyActive := FALSE;
    S_SafetyRequest := FALSE;
    Error := FALSE;
16#8002:
    Ready := TRUE;
    S_SafetyActive := FALSE;
    S_SafetyRequest := TRUE;
    Error := FALSE;
16#8003:
    Ready := TRUE;
    S_SafetyActive := FALSE;
    S_SafetyRequest := FALSE;
    Error := FALSE;
16#8005:
    Ready := TRUE;
    S_SafetyActive := FALSE;
    S_SafetyRequest := FALSE;
    Error := FALSE;
16#8012:
    Ready := TRUE;
    S_SafetyActive := FALSE;
    S_SafetyRequest := TRUE;
    Error := FALSE;
16#C002:
    Ready := TRUE;
    S_SafetyActive := FALSE;
    S_SafetyRequest := FALSE;
    Error := TRUE;
16#C003:
    Ready := TRUE;
    S_SafetyActive := FALSE;
    S_SafetyRequest := FALSE;
    Error := TRUE;
16#C004:
    Ready := TRUE;
    S_SafetyActive := FALSE;
    S_SafetyRequest := FALSE;
    Error := TRUE;
16#C005:
    Ready := TRUE;
    S_SafetyActive := FALSE;
    S_SafetyRequest := FALSE;
    Error := TRUE;
END_CASE;

END_FUNCTION_BLOCK;

(* ---- twoHandControl_II_X.st ---- *)
FUNCTION_BLOCK SF_TwoHandControlTypeII2
 VAR_INPUT
        Activate       : BOOL := FALSE;
        S_Button1      : SAFEBOOL := FALSE;
        S_Button2      : SAFEBOOL := FALSE;
 END_VAR
 VAR_OUTPUT
        Ready          : BOOL := FALSE;
        S_TwoHandOut   : BOOL := FALSE;
        Error          : BOOL := FALSE;
        DiagCode       : WORD := 16#0;
 END_VAR

 IF NOT Activate THEN
     DiagCode := 16#0000;
 ELSE

 CASE DiagCode OF
 16#0000:
     IF Activate THEN
          DiagCode := 16#8001;
     END_IF;

 16#8001:
     IF S_Button1 AND S_Button2 THEN
	     DiagCode := 16#C003;
     ELSIF S_Button1 THEN
	     DiagCode := 16#C001;
	 ELSIF S_Button2 THEN
	     DiagCode := 16#C002;
     ELSE
	     DiagCode := 16#8004;
     END_IF;
 16#8004:
     IF S_Button1 AND S_Button2 THEN
	     DiagCode := 16#8000;
     ELSIF S_Button1 THEN
	     DiagCode := 16#8005;
	 ELSIF S_Button2 THEN
	     DiagCode := 16#8006;
	 END_IF;
 16#8005:
     IF NOT (S_Button1 OR S_Button2) THEN
	     DiagCode := 16#8004;
	 ELSIF NOT S_Button1 AND S_Button2 THEN
	     DiagCode := 16#8019;
	 ELSIF S_Button1 AND S_Button2 THEN
	     DiagCode := 16#8000;
     END_IF;
 16#8006:
     IF NOT (S_Button1 OR S_Button2) THEN
	     DiagCode := 16#8004;
     ELSIF S_Button1 AND NOT S_Button2 THEN
	     DiagCode := 16#8019;
	 ELSIF S_Button1 AND S_Button2 THEN
	     DiagCode := 16#8000;
     END_IF;
 16#8007:
     IF S_Button1 AND S_Button2 THEN
	     DiagCode := 16#8009;
	 ELSIF NOT S_Button1 AND S_Button2 THEN
	     DiagCode := 16#8008;
	 ELSIF NOT (S_Button1 OR S_Button2) THEN
	     DiagCode := 16#8004;
	 END_IF;
 16#8008:
     IF S_Button1 AND S_Button2 THEN
         DiagCode := 16#8009;
     ELSIF S_Button1 AND NOT S_Button2 THEN
	     DiagCode := 16#8007;
     ELSIF NOT (S_Button1 OR S_Button2) THEN
	     DiagCode := 16#8004;
	 END_IF;
 16#8009:
     IF NOT S_Button1 AND S_Button2 THEN
	    DiagCode := 16#8008;
	 ELSIF S_Button1 AND NOT S_Button2 THEN
	     DiagCode := 16#8007;
	 ELSIF NOT (S_Button1 OR S_Button2) THEN
	     DiagCode := 16#8004;
	 END_IF;
 16#8019:
     IF NOT (S_Button1 OR S_Button2) THEN
	     DiagCode := 16#8004;
     END_IF;
 16#8000:
     IF S_Button1 AND NOT S_Button2 THEN
	     DiagCode := 16#8007;
	 ELSIF NOT S_Button1 AND S_Button2 THEN
	     DiagCode := 16#8008;
	 ELSIF NOT (S_Button1 OR S_Button2) THEN
	     DiagCode := 16#8004;
	 END_IF;
 16#C001,
 16#C002,
 16#C003:
     IF NOT (S_Button1 OR S_Button2) THEN
	     DiagCode := 16#8004;
	 END_IF;

 END_CASE;
 END_IF;

 CASE DiagCode OF
  16#0000:
      Ready := FALSE;
      ERROR := FALSE;
      S_TwoHandOut := FALSE;
 16#8000:
      Ready := TRUE;
      ERROR := FALSE;
      S_TwoHandOut := TRUE;
 16#8001,
 16#8004,
 16#8005,
 16#8006,
 16#8007,
 16#8008,
 16#8009,
 16#8019:
      Ready := TRUE;
      ERROR := FALSE;
      S_TwoHandOut := FALSE;
 16#C001,
 16#C002,
 16#C003:
      Ready := TRUE;
      ERROR := TRUE;
      S_TwoHandOut := FALSE;
 END_CASE;

END_FUNCTION_BLOCK

(* ---- twohandControl_III_X.st ---- *)
FUNCTION_BLOCK SF_TwoHandControlTypeIII2
 VAR_INPUT
    Activate          : BOOL;
    S_Button1         : SAFEBOOL;
    S_Button2         : SAFEBOOL;
 END_VAR

 VAR_OUTPUT
    Ready             : BOOL;
    S_TwoHandOut      : SAFEBOOL;
    Error             : BOOL;
    DiagCode          : WORD:=16#0000;
 END_VAR

 VAR
    T_1: TONX;
 END_VAR

IF NOT Activate THEN
    DiagCode := 16#0000;
ELSE

CASE DiagCode OF
16#0000:
    IF Activate THEN
        DiagCode := 16#8001;
    END_IF;
16#8000:
    IF S_Button1 AND NOT S_Button2 THEN
        DiagCode := 16#8007;
    ELSIF NOT S_Button1 AND S_Button2 THEN
        DiagCode := 16#8008;
    ELSIF NOT (S_Button1 OR S_Button2) THEN
        DiagCode := 16#8004;
    END_IF;
16#8001:
    IF S_Button1 AND S_Button2 THEN
        DiagCode := 16#C003;
    ELSIF S_Button1 THEN
        DiagCode := 16#C001;
    ELSIF S_Button2 THEN
        DiagCode := 16#C002;
    ELSIF NOT (S_Button1 OR S_Button2) THEN
        DiagCode := 16#8004;
    END_IF;
16#8004:
    IF S_Button1 AND S_Button2 THEN
        DiagCode := 16#8000;
    ELSIF S_Button1 THEN
        DiagCode := 16#8005;
    ELSIF S_Button2 THEN
        DiagCode := 16#8006;
    END_IF;
16#8005:
    IF T_1.Q THEN
        IF S_Button1 AND S_Button2 THEN
            DiagCode := 16#C006;
        ELSIF S_Button1 THEN
            DiagCode := 16#C005;
        ELSIF S_Button2 THEN
            DiagCode := 16#C004;
        END_IF;
    ELSIF NOT (S_Button1 OR S_Button2) THEN
        DiagCode := 16#8004;
    ELSIF NOT S_Button1 AND S_Button2 THEN
        DiagCode := 16#8019;
    ELSIF S_Button1 AND S_Button2 THEN
        DiagCode := 16#8000;
    END_IF;
16#8006:
    IF T_1.Q THEN
        IF S_Button1 AND S_Button2 THEN
            DiagCode := 16#C006;
        ELSIF S_Button1 THEN
            DiagCode := 16#C005;
        ELSIF S_Button2 THEN
            DiagCode := 16#C004;
        END_IF;
    ELSIF NOT (S_Button1 OR S_Button2) THEN
        DiagCode := 16#8004;
    ELSIF S_Button1 AND NOT S_Button2 THEN
        DiagCode := 16#8019;
    ELSIF S_Button1 AND S_Button2 THEN
        DiagCode := 16#8000;
    END_IF;
16#8007:
    IF S_Button1 AND S_Button2 THEN
        DiagCode := 16#8009;
    ELSIF NOT S_Button1 AND S_Button2 THEN
        DiagCode := 16#8008;
    ELSIF NOT (S_Button1 OR S_Button2) THEN
        DiagCode := 16#8004;
    END_IF;
16#8008:
    IF S_Button1 AND S_Button2 THEN
        DiagCode := 16#8009;
    ELSIF S_Button1 AND NOT S_Button2 THEN
        DiagCode := 16#8007;
    ELSIF NOT (S_Button1 OR S_Button2) THEN
        DiagCode := 16#8004;
    END_IF;
16#8009:
    IF NOT S_Button1 AND S_Button2 THEN
        DiagCode := 16#8008;
    ELSIF S_Button1 AND NOT S_Button2 THEN
        DiagCode := 16#8007;
    ELSIF NOT (S_Button1 OR S_Button2) THEN
        DiagCode := 16#8004;
    END_IF;
16#8019:
    IF NOT (S_Button1 OR S_Button2) THEN
        DiagCode := 16#8004;
    END_IF;
16#C001,
16#C002,
16#C003,
16#C004,
16#C005,
16#C006:
    IF NOT (S_Button1 OR S_Button2) THEN
        DiagCode := 16#8004;
    END_IF;
END_CASE;
END_IF;

IF DiagCode = 16#8005 OR DiagCode = 16#8006 THEN
T_1(IN:=1, PT:=TIME#500ms);
ELSE
T_1(IN:=0, PT:=TIME#500ms);
END_IF;

CASE DiagCode OF
16#0000:
    Ready := FALSE;
    S_TwoHandOut := FALSE;
    Error := FALSE;
16#8000:
    Ready := TRUE;
    S_TwoHandOut := TRUE;
    Error := FALSE;
16#8001,
16#8004,
16#8005,
16#8006,
16#8007,
16#8008,
16#8009,
16#8019:
    Ready := TRUE;
    S_TwoHandOut := FALSE;
    Error := FALSE;
16#C001,
16#C002,
16#C003,
16#C004,
16#C005,
16#C006:
    Ready := TRUE;
    S_TwoHandOut := FALSE;
    Error := TRUE;
END_CASE;

END_FUNCTION_BLOCK

(* ---- 4.1.DiagnosticsConcept.st ---- *)
PROGRAM DiagnosticsConcept
USING PLCopenX;

  VAR_INPUT
	S1_S_EStopIn_1 : SAFEBOOL;
	S1_S_EStopIn_2 : SAFEBOOL;
	S2_S_ESPE_In : SAFEBOOL;
	S0_Reset : BOOL;
	S3_Drive_Reset : BOOL;
	AxisD_1 : INT;
	InputDevice1_active : BOOL;
	InputDevice2_active : BOOL;
	Internal_Acknowledge: BOOL;
  END_VAR
  VAR_OUTPUT
    Error_Equiv1 : BOOL;
	Diag_Equiv1 : WORD;
	Error_EStop1 : BOOL;
	Diag_EStop1 : WORD;
	Error_ESPE1 : BOOL;
	Diag_ESPE1 : WORD;
	Error_SafeStop1 : BOOL;
	Diag_SafeStop1 : WORD;
    S_Stopped : BOOL;
  END_VAR
  VAR
  	S_EStopOut : SAFEBOOL;
	SF_Equivalent_1 : SF_EquivalentX;
	SF_EmergencyStop_1 : SF_EmergencyStopX;
	SF_ESPE_1 : SF_ESPEX;
	SF_SafeStop1_1 : SF_SafeStop1X;
  END_VAR

  SF_Equivalent_1(InputDevice1_active, S1_S_EStopIn_1, S1_S_EStopIn_2, T#10ms);
  SF_EmergencyStop_1(SF_Equivalent_1.Ready, SF_Equivalent_1.S_EquivalentOut, FALSE, FALSE, S0_Reset);
  SF_ESPE_1(InputDevice2_active, S2_S_ESPE_In, FALSE, FALSE, S0_Reset);
  SF_SafeStop1_1(
    Activate:=SF_EmergencyStop_1.Ready AND SF_ESPE_1.Ready,
    S_StopIn:=S_EStopOut AND SF_ESPE_1.S_ESPE_Out,
    AxisID:=AxisD_1,
    MonitoringTime:=T#100ms,
    Reset:=S3_Drive_Reset,
    Acknowledge := Internal_Acknowledge);
  S_EStopOut := SF_EmergencyStop_1.S_EStopOut;
  Error_Equiv1 := SF_Equivalent_1.Error;
  Diag_Equiv1 := SF_Equivalent_1.DiagCode;
  Error_EStop1 := SF_EmergencyStop_1.Error;
  Diag_EStop1 := SF_EmergencyStop_1.DiagCode;
  Error_ESPE1 := SF_ESPE_1.Error;
  Diag_ESPE1 := SF_ESPE_1.DiagCode;
  Error_SafeStop1 := SF_SafeStop1_1.Error;
  Diag_SafeStop1 := SF_SafeStop1_1.DiagCode;
  S_Stopped := SF_SafeStop1_1.S_Stopped;
END_PROGRAM

(* ---- RTAndroid_flagDelayAsInput.st ---- *)
PROGRAM cyclic
(* Moegliche Zustaende fuer den Automaten *)
VAR CONSTANT
	stateAfterBoot : BYTE := 0;
	stateInit : BYTE := 1;
	stateWaitForItem : BYTE := 2;
	stateWaitForCompressor1 : BYTE := 3;
	stateExtractItem1 : BYTE := 4;
	stateWaitForCompressor2 : BYTE := 5;
	stateExtractItem2 : BYTE := 6;
	stateRotateTable1 : BYTE := 7;
	stateWaitForCompressor3 : BYTE := 8;
	statePunchItem : BYTE := 9;
	stateRotateTable2 : BYTE := 10;
	stateWaitForCompressor4 : BYTE := 11;
	stateMoveToConveyer1 : BYTE := 12;
	stateWaitForCompressor5 : BYTE := 13;
	stateMoveToConveyer2 : BYTE := 14;
	stateRunConveyer : BYTE := 15;
	stateMoveToRobot : BYTE := 16;
	stateTurnToItem : BYTE := 17;
	stateTakeItem : BYTE := 18;
	stateTurnToMagazin : BYTE := 19;
	stateError : BYTE := 20;
END_VAR
(* Vordefinierte Konstanten fuer den gesamten Ablauf *)
VAR CONSTANT
	pickPosTurn : BYTE := 111;
	pickPosVert : BYTE := 80;
	pickPosArm : BYTE := 28;
	pickPosClaw : BYTE := 19;
	dropPosTurn : BYTE := 71;
	dropPosArm : BYTE := 37;
	moveThreshold : BYTE := 36;
	compressorDelay : DINT := 50;
	extractionDelay : DINT := 50;
	conveyerDelay : DINT := 50;
	waitForItemThreshold : DINT := 100;
	waitForPuncherThreshold : DINT := 10;
END_VAR
(* Virtuelle Speicherstellen der Sensoren / Motoren *)
VAR_INPUT
	(* 3D-Roboter *)
	turnDestPos : BYTE;
	turnCurrPos : BYTE;
	vertDestPos  : BYTE;
	vertCurrPos : BYTE;
	armDestPos  : BYTE;
	armCurrPos   : BYTE;
	clawDestPos  : BYTE;
	clawCurrPos  : BYTE;
	(* Bearbeitungszentrum *)
	compressor : BYTE;
	tableMotPow  : BYTE;
	tableMotDir  : BYTE;
	magazinLed  : BYTE;
	magazinPhoto : BYTE;
	magazinPusherOn  : BYTE;
	magazinPusherOff : BYTE;
	conveyerMotPow  : BYTE;
	conveyerMotDir  : BYTE;
	conveyerLed  : BYTE;
	conveyerPhoto  : BYTE;
	conveyerButton : BYTE;
	conveyerPusherOn  : BYTE;
	conveyerPusherOff  : BYTE;
	puncherButton  : BYTE;
	puncher  : BYTE;

	flagDelay : DINT;
END_VAR

(* Verwendete Ein- und Ausgaenge *)
VAR_OUTPUT
	outState : BYTE;
	outError : BOOL := false;
	DiagCode : BYTE := 16#0000;
END_VAR

	(* Motoren einmalig zur Nullposition fahren *)
	IF DiagCode = stateAfterBoot THEN

		compressor := 0;

		tableMotPow := 0;
		tableMotDir := 0;

		magazinLed := 0;
		magazinPusherOn := 0;
		magazinPusherOff := 0;

		conveyerMotPow := 0;
		conveyerMotDir := 0;
		conveyerLed := 0;
		conveyerPusherOn := 0;
		conveyerPusherOff := 0;

		turnDestPos := 0;
		vertDestPos := 0;
		armDestPos := 0;
		clawDestPos := 0;

		IF turnCurrPos = 0 AND armCurrPos = 0 AND clawCurrPos = 0 THEN
			DiagCode := stateInit;
		END_IF

	(* Anlage vor dem Start initialisieren *)
	ELSIF DiagCode = stateInit THEN

		conveyerLed := 1;
		magazinLed := 1;

		turnDestPos := dropPosTurn;
		armDestPos := dropPosArm;

		IF turnCurrPos = dropPosTurn AND armCurrPos = dropPosArm AND vertCurrPos = 0 THEN
			IF clawCurrPos = 0 THEN
				DiagCode := stateWaitForItem;
			ELSE
				clawDestPos := 0;
			END_IF
		END_IF

	(* Warten, bis sich ein Werkstueck im Magazin befindet *)
	ELSIF DiagCode = stateWaitForItem THEN

		IF flagDelay = waitForItemThreshold THEN
			DiagCode := stateInit;
		ELSIF magazinPhoto = 1 THEN
			magazinLed := 0;
			DiagCode := stateWaitForCompressor1;
		END_IF

	(* Kompressor zum Ausfahren des Magazinschiebers vorbereiten *)
	ELSIF DiagCode = stateWaitForCompressor1 THEN

		compressor := 1;

		IF flagDelay >= compressorDelay THEN
			compressor := 0;
			DiagCode := stateExtractItem1;
		END_IF

	(* Werkstueck aus dem Magazin entnehmen - Teil 1 *)
	ELSIF DiagCode = stateExtractItem1 THEN

		magazinPusherOn := 1;

		IF flagDelay >= extractionDelay THEN
			magazinPusherOn := 0;
			DiagCode := stateWaitForCompressor2;
		END_IF

	(* Kompressor zum Einfahren des Magazinschiebers vorbereiten *)
	ELSIF DiagCode = stateWaitForCompressor2 THEN

		compressor := 1;

		IF flagDelay >= compressorDelay THEN
			compressor := 0;
			DiagCode := stateExtractItem2;
		END_IF

	(* Werkstueck aus dem Magazin entnehmen - Teil 2 *)
	ELSIF DiagCode = stateExtractItem2 THEN

		magazinPusherOff := 1;

		IF flagDelay >= extractionDelay THEN
			magazinPusherOff := 0;
			DiagCode := stateRotateTable1;
		END_IF

	(* Drehtisch aktivieren und Stanze-Schalter ueberwachen *)
	ELSIF DiagCode = stateRotateTable1 THEN

		tableMotPow := 200;
		(* something went wrong: we skip punching *)
		IF flagDelay > waitForPuncherThreshold THEN
			tableMotPow := 0;
			DiagCode := stateRotateTable2;
		ELSIF puncherButton = 0 THEN
			tableMotPow := 0;
			DiagCode := stateWaitForCompressor3;
		END_IF

	(* Kompressor zum Stanzen vorbereiten *)
	ELSIF DiagCode = stateWaitForCompressor3 THEN

		compressor := 1;

		IF flagDelay >= compressorDelay THEN
			compressor := 0;
			DiagCode := statePunchItem;
		END_IF

	(* Werkstueck stanzen *)
	ELSIF DiagCode = statePunchItem THEN

		puncher := 1;

		IF flagDelay >= extractionDelay THEN
			puncher := 0;
			DiagCode := stateRotateTable2;
		END_IF

	(* Drehtisch aktivieren und Transportband-Schalter ueberwachen *)
	ELSIF DiagCode = stateRotateTable2 THEN

		tableMotPow := 200;

		IF conveyerButton = 0 THEN
			tableMotPow := 0;
			DiagCode := stateWaitForCompressor4;
		END_IF
	(* Kompressor zum Einfahren des Transportschiebers vorbereiten *)
	ELSIF DiagCode = stateWaitForCompressor4 THEN

		compressor := 1;

		IF flagDelay >= compressorDelay THEN
			compressor := 0;
			DiagCode := stateMoveToConveyer1;
		END_IF

	(* Werkstueck auf das Fliessband befoerdern - Teil 1 *)
	ELSIF DiagCode = stateMoveToConveyer1 THEN

		conveyerPusherOn := 1;

		IF flagDelay >= extractionDelay THEN
			conveyerPusherOn := 0;
			DiagCode := stateWaitForCompressor5;
		END_IF

	(* Kompressor zum Ausfahren des Transportschiebers vorbereiten *)
	ELSIF DiagCode = stateWaitForCompressor5 THEN

		compressor := 1;

		IF flagDelay >= compressorDelay THEN
			compressor := 0;
			DiagCode := stateMoveToConveyer2;
		END_IF

	(* Werkstueck auf das Fliessband befoerdern - Teil 2 *)
	ELSIF DiagCode = stateMoveToConveyer2 THEN

		conveyerPusherOff := 1;

		IF flagDelay >= extractionDelay THEN
			conveyerPusherOff := 0;
			DiagCode := stateRunConveyer;
		END_IF

	(* Fliessband aktivieren und auf das Werkstueck warten *)
	ELSIF DiagCode = stateRunConveyer THEN

		conveyerMotPow := 200;
		(*Something went wrong, we again try to put the item on the tape *)
		IF flagDelay = waitForItemThreshold THEN
			DiagCode := stateMoveToConveyer1;
		ELSIF conveyerPhoto = 1 THEN
			conveyerLed := 0;
			DiagCode := stateMoveToRobot;
		END_IF

	(* Drehen, Greifarm und Greifer ausstrecken *)
	ELSIF DiagCode = stateMoveToRobot THEN

		IF flagDelay > conveyerDelay THEN
			conveyerMotPow := 0;
			DiagCode := stateTurnToItem;
		END_IF

	(* Drehen, Greifarm und Greifer ausstrecken *)
	ELSIF DiagCode = stateTurnToItem THEN

		turnDestPos := pickPosTurn;
		vertDestPos := pickPosVert;
		armDestPos := pickPosArm;

		IF turnCurrPos = pickPosTurn AND vertCurrPos = pickPosVert AND armCurrPos = pickPosArm THEN
			DiagCode := stateTakeItem;
		END_IF

	(* Werkstueck vom Fliessband greifen *)
	ELSIF DiagCode = stateTakeItem THEN

		clawDestPos := pickPosClaw;

		IF clawCurrPos = pickPosClaw THEN
			DiagCode := stateTurnToMagazin;
		END_IF

	(* Das Werkstueck zum Magazin drehen *)
	ELSIF DiagCode = stateTurnToMagazin THEN

		vertDestPos := 0;

		IF vertCurrPos < moveThreshold THEN
			DiagCode := stateInit;
		END_IF

	(* Fehlerzustand - alles ausschalten *)
	ELSE

		outError := true;

		compressor := 0;
		puncher := 0;

		tableMotPow := 0;
		tableMotDir := 2;

		conveyerMotPow := 0;
		conveyerMotDir := 2;

	(* Ende des Zustandsautomaten *)
	END_IF

	(* Ausgabe vorbereiten *)
	outState := DiagCode;

END_PROGRAM
